// Mitsubishi GX Works2 project: 타이머 점멸 답안   PLC: Q03UDV

PROGRAM MAIN
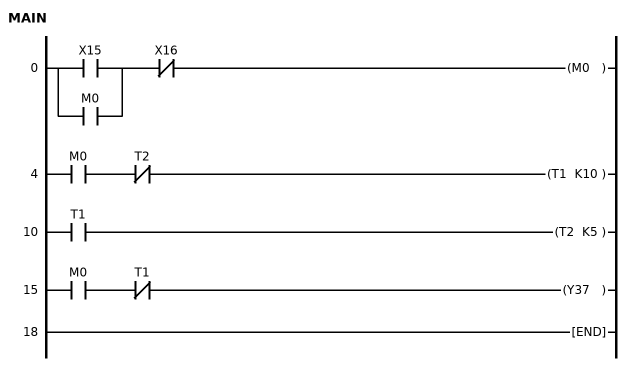
0     LD      X15
      OR      M0
      ANI     X16
      OUT     M0
4     LD      M0
      ANI     T2
      OUT     T1 K10
10    LD      T1
      OUT     T2 K5
15    LD      M0
      ANI     T1
      OUT     Y37
18    END
END_PROGRAM
